(* IEC 61131-3 sources: AXOpen/src/timers/ctrl/src, 4 files *)

(* ---- AxoBlinker.st ---- *)
USING AXOpen.Core;

NAMESPACE AXOpen.Timers

    ///<summary>
    /// Provides periodic on/off switcher.
    ///</summary>
    {S7.extern=ReadWrite}
    CLASS AxoBlinker
        VAR PUBLIC
            output : BOOL;
        END_VAR

        VAR PRIVATE
            _onTimer    : OnDelayTimer;
            _offTimer   : OnDelayTimer;

            _nextExpectedCycle : ULINT;
            _state : INT;
        END_VAR

        ///<summary>
        /// Provides periodic on/off switcher.
        ///</summary>
        METHOD PUBLIC Blink : BOOL
            VAR_INPUT
                Parent : IAxoObject;
                ///<summary>
                /// Time duration for on duty output.
                ///</summary>
                inOnTime : TIME;
                ///<summary>
                /// Time duration for off duty output.
                ///</summary>
                inOffTime : TIME;
            END_VAR

            IF Parent = NULL THEN
                RETURN;
            END_IF;

            Blink := THIS.Execute(Parent,inOnTime,inOffTime);
        END_METHOD

        ///<summary>
        /// Provides periodic on/off switcher.
        ///</summary>
        METHOD PUBLIC Blink : BOOL
            VAR_INPUT
                Context : IAxoContext;
                ///<summary>
                /// Time duration for on duty output.
                ///</summary>
                inOnTime : TIME;
                ///<summary>
                /// Time duration for off duty output.
                ///</summary>
                inOffTime : TIME;
            END_VAR

            IF Context = NULL THEN RETURN; END_IF;
            IF(Context.GetRtm() = NULL) THEN RETURN; END_IF;

            Blink := THIS.Execute(Context,inOnTime,inOffTime);
        END_METHOD

        METHOD PRIVATE Execute : BOOL
            VAR_INPUT
                Context : IAxoContext;
                inOnTime : TIME;
                inOffTime : TIME;
            END_VAR

            IF( Context.OpenCycleCount() <>  _nextExpectedCycle) THEN
                _state := 0;
            END_IF;

            _nextExpectedCycle := Context.OpenCycleCount() + ULINT#1;

            IF(_state = 0) THEN
                _offTimer.OnDelay(Context := Context, inSignal := FALSE, TimeDelay := T#0S);
                 _onTimer.OnDelay(Context := Context, inSignal := FALSE, TimeDelay := T#0S);
                _state := 1;
            END_IF;

            IF(_state = 1) THEN
                output := TRUE;
                IF(_onTimer.OnDelay(Context := Context ,inSignal := TRUE, TimeDelay:=inOnTime)) THEN
                    _state := 2;
                    RETURN;
                END_IF;
            END_IF;

            IF(_state = 2) THEN
                output := FALSE;
                IF(_offTimer.OnDelay(Context := Context, inSignal := TRUE, TimeDelay:=inOffTime)) THEN
                    _state := 0;
                END_IF;
            END_IF;
        END_METHOD

        METHOD PRIVATE Execute : BOOL
            VAR_INPUT
                Parent : IAxoObject;
                inOnTime : TIME;
                inOffTime : TIME;
            END_VAR

            IF( Parent.GetContext().OpenCycleCount() <>  _nextExpectedCycle) THEN
                _state := 0;
            END_IF;

            _nextExpectedCycle := Parent.GetContext().OpenCycleCount() + ULINT#1;

            IF(_state = 0) THEN
                _offTimer.OnDelay(Parent := Parent,inSignal := FALSE, TimeDelay:=T#0S);
                _onTimer.OnDelay(Parent := Parent,inSignal := FALSE, TimeDelay:=T#0S);
                _state := 1;
            END_IF;

            IF(_state = 1) THEN
                output := TRUE;
                IF(_onTimer.OnDelay(Parent:= Parent ,inSignal := TRUE, TimeDelay:=inOnTime)) THEN
                    _state := 2;
                    RETURN;
                END_IF;
            END_IF;

            IF(_state = 2) THEN
                output := FALSE;
                IF(_offTimer.OnDelay(Parent := Parent,inSignal := TRUE, TimeDelay:=inOffTime)) THEN
                    _state := 0;
                END_IF;
            END_IF;
        END_METHOD

        ///<summary>
        /// Method for restoring default values of blinker.
        ///</summary>
        METHOD PUBLIC Restore
            _onTimer.Restore();
            _offTimer.Restore();
            _nextExpectedCycle := ULINT#0;
            _state := INT#0;
            output := FALSE;
        END_METHOD
    END_CLASS
END_NAMESPACE

(* ---- OffDelay.st ---- *)
USING AXOpen.Core;

NAMESPACE AXOpen.Timers

    ///<summary>
    /// OffDelayTimer class, which contains OffDelay method representing timer.
    /// Counting of timer start on FALLING edge.
    ///</summary>
    {S7.extern=ReadWrite}
    CLASS OffDelayTimer
        VAR PUBLIC
            output : BOOL;
            elapsedTime : LTIME;
        END_VAR

        VAR PRIVATE
          _startTime : LTIME;
          _previousSignalStatus : BOOL;
          _currentTimeDiff : LTIME;
          _isCounting : BOOL;

        END_VAR

        ///<summary>
        /// OffDelay timer, which output it FALSE when time delay is counted, otherwise always returns TRUE.
        /// Counting of timer start on FALLING edge.
        /// IAxoObject is used to acquire context automatically.
        ///</summary>
        METHOD PUBLIC OffDelay : BOOL
            VAR_INPUT
                Parent : IAxoObject;
                inSignal : BOOL;
                TimeDelay : LTIME;
            END_VAR
            OffDelay := THIS.OffDelay(Parent.GetContext(), inSignal, TimeDelay);
        END_METHOD

        ///<summary>
        /// OffDelay timer, which output it FALSE when time delay is counted, otherwise always returns TRUE.
        /// Counting of timer start on FALLING edge.
        /// IAxoContext is directly required.
        ///
        /// When IN is TRUE, Q is TRUE and ET is 0.
        /// As soon as IN becomes FALSE, the time will begin to be counted in milliseconds in ET until its value is equal to that of PT.
        /// It will then remain constant.
        /// Q is FALSE when IN is FALSE and ET is equal to PT.
        /// Otherwise it is TRUE.
        /// Thus, Q has a falling edge when the time indicated in PT in milliseconds has run out.
        ///</summary>
        METHOD PUBLIC OffDelay : BOOL
            VAR_INPUT
                Context : IAxoContext;
                inSignal : BOOL;
                TimeDelay : LTIME;
            END_VAR

            IF(Context = NULL) THEN RETURN; END_IF;

            // if input signal is off and previous signal was off, no edge detected, return output false
            IF(NOT inSignal AND NOT THIS._previousSignalStatus) THEN
                OffDelay := FALSE;
                output := OffDelay;
                THIS._previousSignalStatus := inSignal;
                RETURN;
            END_IF;

            // RISING EDGE detected, set output to true
            // if inSignal is true, and previous is false, set output to true
            // restore timer on rising edge
            IF(inSignal AND NOT THIS._previousSignalStatus) THEN
                THIS.Restore();
                OffDelay := TRUE;
                output := OffDelay;
                THIS._previousSignalStatus := inSignal;
                RETURN;
            END_IF;

           // FALLING EDGE  detected start timer counting
           // start computing on falling edge (if actual signal is false, but previous was true)
            IF(NOT inSignal AND THIS._previousSignalStatus) THEN
                THIS._startTime := Context.GetRtm().Elapsed();
                _isCounting := TRUE;
            END_IF;

            // if timer is counting, compute difference and watch for end of timer
            IF(THIS._isCounting) THEN
                _currentTimeDiff := Context.GetRtm().Elapsed() - THIS._startTime ;
                // if timer passed, set output to false
                OffDelay := NOT (_currentTimeDiff >= TimeDelay);
                output := OffDelay;
                elapsedTime :=  _currentTimeDiff;
                THIS._previousSignalStatus := inSignal;

            ELSE
                // here timer is not counting, therefore output will be set to true
                // I get here, when previousSignal was true, and actual signal is still true
                OffDelay := TRUE;
                output := OffDelay;
                elapsedTime :=  LTIME#0s;
                THIS._previousSignalStatus := inSignal;
            END_IF;

        END_METHOD

        ///<summary>
        /// Method for restoring default values of timer.
        ///</summary>
        METHOD PUBLIC Restore
            _isCounting := FALSE;
            _previousSignalStatus := FALSE;
            _currentTimeDiff := LTIME#0s;
            _startTime := LTIME#00H00M00S0MS0NS;
        END_METHOD

    END_CLASS
END_NAMESPACE

(* ---- OnDelay.st ---- *)
USING AXOpen.Core;

NAMESPACE AXOpen.Timers

    ///<summary>
    /// OnDelayTimer class, which contains OnDelay method representing timer.
    /// Counting of timer start on RISING edge.
    ///</summary>
    {S7.extern=ReadWrite}
    CLASS OnDelayTimer
        VAR PUBLIC
            output : BOOL;
            elapsedTime : LTIME;
        END_VAR

        VAR PRIVATE
          _startTime : LTIME;
          _previousSignalStatus : BOOL;
          _currentTimeDiff : LTIME;

        END_VAR

        ///<summary>
        /// OnDelay timer, which output is TRUE when time delay is counted, otherwise always returns FALSE.
        /// Counting of timer start on RISING edge.
        ///</summary>
        METHOD PUBLIC OnDelay : BOOL
            VAR_INPUT
                Parent : IAxoObject;
                inSignal : BOOL;
                TimeDelay : LTIME;
            END_VAR

            OnDelay := THIS.OnDelay(Parent.GetContext(), inSignal, TimeDelay);
        END_METHOD

        /// LOGIC OF ONDELAY TIMER
        /// If IN is FALSE, Q is FALSE and ET is 0.
        /// As soon as IN becomes TRUE, the time will begin to be counted in milliseconds in ET until its value is equal to PT.
        /// It will then remain constant. Q is TRUE when IN is TRUE and ET is equal to PT.
        /// Otherwise it is FALSE.
        /// Thus, Q has a rising edge when the time indicated in PT in milliseconds has run out.

        ///<summary>
        /// OnDelay timer, which output is TRUE when time delay is counted, otherwise always returns FALSE.
        /// Counting of timer start on RISING edge.
        ///</summary>
        METHOD PUBLIC OnDelay : BOOL
            VAR_INPUT
                Context : IAxoContext;
                inSignal : BOOL;
                TimeDelay : LTIME;
            END_VAR

            IF(Context = NULL) THEN RETURN; END_IF;
            IF(Context.GetRtm() = NULL) THEN RETURN; END_IF;

            // beggining, if all is turn off, return false
            IF(NOT inSignal AND NOT THIS._previousSignalStatus) THEN
                OnDelay := FALSE;
                output := OnDelay;
                elapsedTime := LTIME#0s;
                RETURN;
            END_IF;

            // start counting on RISING edge
            // start counting when inputSignal is true and previous signal was not set
            IF(inSignal AND NOT THIS._previousSignalStatus) THEN
                THIS._startTime := Context.GetRtm().Elapsed();
            END_IF;

            // FALLING edge detected
            // if input signal is turned off and previous signal was true, that means output must by false, we do not need to compute time
            // let's afterwards restore timer to default values
            IF(NOT inSignal AND THIS._previousSignalStatus) THEN
                THIS.Restore();
                THIS._previousSignalStatus := inSignal;
                OnDelay := FALSE;
                output := OnDelay;
                elapsedTime := _currentTimeDiff;

                RETURN;
            END_IF;

            _currentTimeDiff := Context.GetRtm().Elapsed() - THIS._startTime ;
            OnDelay := _currentTimeDiff >= TimeDelay;
            output := OnDelay;
            elapsedTime :=  _currentTimeDiff;
            THIS._previousSignalStatus := inSignal;

        END_METHOD

        ///<summary>
        /// Method for restoring default values of timer.
        ///</summary>
        METHOD PUBLIC Restore
            _previousSignalStatus := FALSE;
            _currentTimeDiff := LTIME#0s;
        END_METHOD

    END_CLASS
END_NAMESPACE

(* ---- Pulse.st ---- *)
USING AXOpen.Core;

NAMESPACE AXOpen.Timers

    ///<summary>
    /// PulseTimer class, which contains Pulse method representing timer.
    /// Counting of timer start on RISING edge.
    ///</summary>
    {S7.extern=ReadWrite}
    CLASS PulseTimer
        VAR PUBLIC
            output : BOOL;
            elapsedTime : LTIME;
        END_VAR

        VAR PRIVATE
          _startTime : LTIME;
          _previousSignalStatus : BOOL;
          _currentTimeDiff : LTIME;

        END_VAR

        METHOD PUBLIC Pulse : BOOL
            VAR_INPUT
                Parent : IAxoObject;
                inSignal : BOOL;
                PulseLenght : LTIME;
            END_VAR
            Pulse := THIS.Pulse(Parent.GetContext(), inSignal, PulseLenght);
        END_METHOD

        ///<summary>
        /// Pulse timer, which output is TRUE only during time counting.
        /// Counting of timer start on RISING edge.
        ///
        /// If IN is FALSE, the outputs are FALSE or 0.
        /// As soon as IN becomes TRUE, Q also becomes TRUE and remains TRUE for the pulse duration PT.
        /// As long as Q is TRUE, the time is incremented in milliseconds in ET, until the value reaches PT.
        /// The value then remains constant.
        /// The output Q remains TRUE until the pulse duration has elapsed, irrespective of the state of the input IN.
        /// Q therefore supplies a signal over the interval specified in PT.
        ///</summary>
        METHOD PUBLIC Pulse : BOOL
            VAR_INPUT
                Context : IAxoContext;
                inSignal : BOOL;
                PulseLenght : LTIME;
            END_VAR

            IF(Context = NULL) THEN
                RETURN;
            END_IF;
            IF(Context.GetRtm() = NULL) THEN
                RETURN;
            END_IF;

            // always, when input is false, outputs are false
            IF(NOT inSignal ) THEN
                Pulse := FALSE;
                output := Pulse;
                elapsedTime := _currentTimeDiff;
                RETURN;
            END_IF;

            // start counting on RISING edge
            // output is true during counting period
            IF(inSignal AND NOT THIS._previousSignalStatus) THEN
                THIS._startTime := Context.GetRtm().Elapsed();
            END_IF;

            _currentTimeDiff := Context.GetRtm().Elapsed() - THIS._startTime ;

            // output is true, if counting is in progress and time diff is smaller then pulse length
            Pulse := _currentTimeDiff < PulseLenght;
            output := Pulse;
            elapsedTime :=  _currentTimeDiff;
            THIS._previousSignalStatus := inSignal;

        END_METHOD

        ///<summary>
        /// Method for restoring default values of timer.
        ///</summary>
        METHOD PUBLIC Restore
            _previousSignalStatus := FALSE;
            _currentTimeDiff := LTIME#0s;
            _startTime := LTIME#00H00M00S000MS0NS;
        END_METHOD

    END_CLASS
END_NAMESPACE
